(* Logix 5000 project; controller PBS_Perfusion vendor 1 type 14 code 217 rev 32.14; software revision 32.03; part 27 of 27 *)
(* tags used below, declared in another part *)
   AIC703 : P_AInAdv;   // BRX DO PV
   AirManualSP : REAL;
   AirPercentOut : REAL;
   AirProgOper : BOOL;
   AT701 : P_AInAdv;   // DO Transmitter
   AT702 : P_AInAdv;   // pH Transmitter
   BRX_Level_EUMax : REAL;
   BRX_Level_EUmin : REAL;
   BRX_Level_Initialize : BOOL;
   BRX_Level_RawMax : REAL;
   BRX_Level_RawMin : REAL;
   CCAMaxCalc : REAL;
   CO2CVMax : REAL;
   CO2CVMin : REAL;
   CO2EUMax : REAL;
   CO2EUMax_Input : REAL;
   CO2EUMin : REAL;
   CO2EUMin_Input : REAL;
   CO2ManualSP : REAL;
   CO2ManualSP_Input : REAL;
   CO2MaxCalc : REAL;
   CO2PercentOut : REAL;
   CO2ProgOper : BOOL;
   conditionedMedia_auto : BOOL;
   ConditionedMedia_Initialize : BOOL;
   CondMedRawMax : REAL;
   CondMedRawMin : REAL;
   DO_HiDev : REAL;   // hi deviation alarm
   DO_LoDev : REAL;   // low deviation alarm
   DO_ON : BOOL;
   DO_PID_AUTOREQ : BOOL;
   DOPID_INITIALIZE : BOOL;
   EStop : P_DIn;
   FIC110 : P_ValveC;   // PBS CCA
   FIC120 : P_ValveC;   // O2 pbs
   FIC130 : P_ValveC;   // CO2 pbs
   FIC140 : P_ValveC;   // pbs N2 mfc
   GasControl_ON : BOOL;
   GasOffOns : BOOL;
   GasOnOns : BOOL;
   Heater_Output : P_AOut;   // Heating blanket AO
   LIT801 : P_AInAdv;   // Level Value From BRX
   ManualDO_CV : REAL;
   ManualpH_CV : REAL;
   N2CVMax : REAL;
   N2CVMin : REAL;
   N2EUMax : REAL;
   N2EUMax_Input : REAL;
   N2EUMin : REAL;
   N2EUMin_Input : REAL;
   N2ManualSP : REAL;
   N2ManualSP_Input : REAL;
   N2MaxCalc : REAL;
   N2PercentOut : REAL;
   N2ProgOper : BOOL;
   O2CVMax : REAL;
   O2CVMin : REAL;
   O2EUMax : REAL;
   O2EUMax_Input : REAL;
   O2EUMin : REAL;
   O2EUMin_Input : REAL;
   O2ManualSP : REAL;
   O2ManualSP_Input : REAL;
   O2MaxCalc : REAL;
   O2PercentOut : REAL;
   O2ProgOper : BOOL;
   ONS : DINT[3];
   P103 : P_VSD;   // Conditioned Media Addition Pump
   Perfusion_Level_Aggression : REAL;
   pH_HiDev : REAL;   // ph hi deviation
   pH_Initialize : BOOL;
   pH_LoDev : REAL;   // pH Lo deviation alarm
   PH_On : BOOL;
   pH_PID_AUTOREQ : BOOL;
   Temp_Initialize : BOOL;
   TempEUMax : REAL;
   TempEUMin : REAL;
   TempOffOns : BOOL;
   TempOnOns : BOOL;
   TempRawMax : REAL;
   TempRawMin : REAL;
   TotalFlowSP : REAL;
   TT700 : P_AInAdv;   // Temperature Transmitter
   TT700_1Point_Complete : BOOL;
   TT700_1Point_Offset : REAL;
   TT700_2Point_Complete : BOOL;
   TT700_2PointAccept : BOOL;
   TT700_Accept1Point : BOOL;
   TT700_CalClear : BOOL;
   TT700_MaxCfg : REAL;
   TT700_MinCfg : REAL;
   TT700_NewMax : REAL;
   TT700_NewMin : REAL;
   TT700_RawMax : REAL;
   TT700_RawMin : REAL;
   TT700_RawRange : REAL;
   TT700_Ref1Point : REAL;
   TT700_RefMax : REAL;
   TT700_RefMin : REAL;
   TT700_RefRange : REAL;
(* CM_PBS, continued *)

ROUTINE RTD_Calibration   (* ladder *)
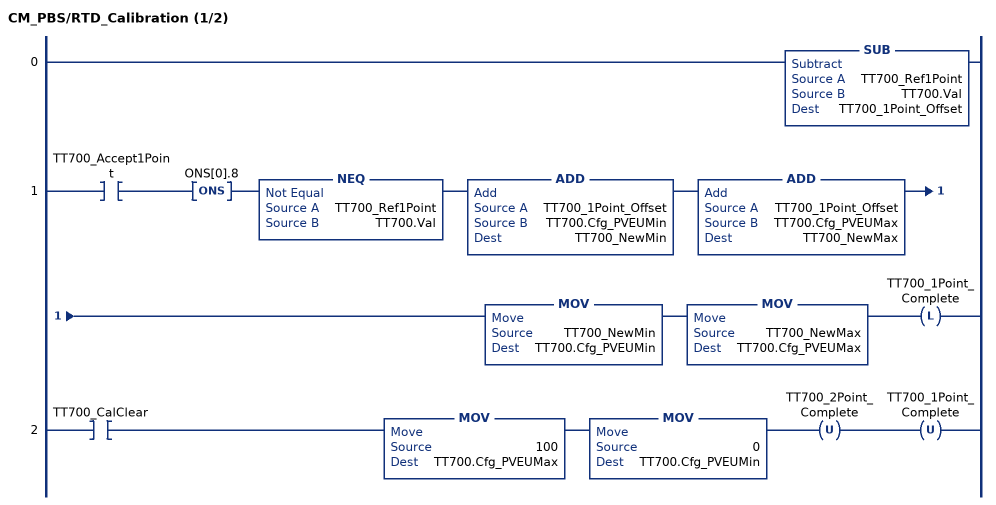
   0: SUB(TT700_Ref1Point,TT700.Val,TT700_1Point_Offset);
   1: XIC(TT700_Accept1Point)ONS(ONS[0].8)NEQ(TT700_Ref1Point,TT700.Val)ADD(TT700_1Point_Offset,TT700.Cfg_PVEUMin,TT700_NewMin)ADD(TT700_1Point_Offset,TT700.Cfg_PVEUMax,TT700_NewMax)MOV(TT700_NewMin,TT700.Cfg_PVEUMin)MOV(TT700_NewMax,TT700.Cfg_PVEUMax)OTL(TT700_1Point_Complete);
   2: XIC(TT700_CalClear)MOV(100,TT700.Cfg_PVEUMax)MOV(0,TT700.Cfg_PVEUMin)OTU(TT700_2Point_Complete)OTU(TT700_1Point_Complete);
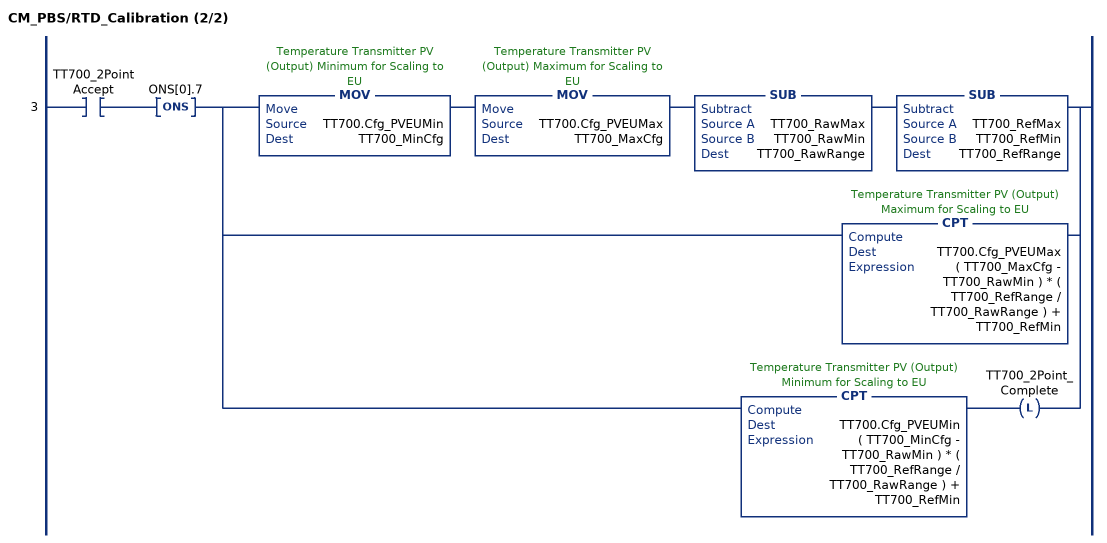
   3: XIC(TT700_2PointAccept)ONS(ONS[0].7)[MOV(TT700.Cfg_PVEUMin,TT700_MinCfg) MOV(TT700.Cfg_PVEUMax,TT700_MaxCfg) SUB(TT700_RawMax,TT700_RawMin,TT700_RawRange) SUB(TT700_RefMax,TT700_RefMin,TT700_RefRange) ,CPT(TT700.Cfg_PVEUMax,( TT700_MaxCfg - TT700_RawMin ) * ( TT700_RefRange / TT700_RawRange ) + TT700_RefMin) ,CPT(TT700.Cfg_PVEUMin,( TT700_MinCfg - TT700_RawMin ) * ( TT700_RefRange / TT700_RawRange ) + TT700_RefMin) OTL(TT700_2Point_Complete) ];
END_ROUTINE
END_PROGRAM

PROGRAM PIDs   (* main routine Main *)
VAR
   ADD_01 : FBD_MATH := (SourceA := 1.0, SourceB := 0.1, Dest := 1.1);
   BOR_01 : FBD_BOOLEAN_OR;
   BOR_02 : FBD_BOOLEAN_OR;
   BOR_03 : FBD_BOOLEAN_OR;
   BOR_04 : FBD_BOOLEAN_OR;
   BOR_05 : FBD_BOOLEAN_OR;
   BOR_06 : FBD_BOOLEAN_OR;
   DIV_01 : FBD_MATH := (SourceA := 10.0, SourceB := 100.0, Dest := 0.1);
   DIV_02 : FBD_MATH := (SourceA := 0.33333334, SourceB := 100.0, Dest := 0.0033333334);
   DIV_03 : FBD_MATH := (SourceB := 100.0);
   DIV_04 : FBD_MATH := (SourceB := 100.0);
   DIV_05 : FBD_MATH := (SourceA := 0.33333334, SourceB := 100.0, Dest := 0.0033333334);
   DIV_06 : FBD_MATH := (SourceA := 0.083333336, SourceB := 100.0, Dest := 0.00083333335);
   DIV_07 : FBD_MATH := (SourceB := 100.0);
   GRT_01 : FBD_COMPARE;
   OSRI_01 : FBD_ONESHOT;
   PIDE_01 : PID_ENHANCED := (PVEUMax := 100.0, SPHLimit := 100.0, RatioProg := 1.0, RatioOper := 1.0, RatioHLimit := 1.0, RatioLLimit := 1.0, CVEUMax := 100.0, CVHLimit := 100.0, PVEDerivative := 1, RTSTime := 1);
   PIDE_02 : PID_ENHANCED := (PVEUMax := 100.0, SPHLimit := 100.0, RatioProg := 1.0, RatioOper := 1.0, RatioHLimit := 1.0, RatioLLimit := 1.0, CVEUMax := 100.0, CVHLimit := 100.0, PVEDerivative := 1, RTSTime := 1);
   PIDE_03 : PID_ENHANCED := (PVEUMax := 100.0, SPHLimit := 100.0, RatioProg := 1.0, RatioOper := 1.0, RatioHLimit := 1.0, RatioLLimit := 1.0, CVEUMax := 100.0, CVHLimit := 100.0, PVEDerivative := 1, RTSTime := 1);
   PIDE_04 : PID_ENHANCED := (PVEUMax := 100.0, SPHLimit := 100.0, RatioProg := 1.0, RatioOper := 1.0, RatioHLimit := 1.0, RatioLLimit := 1.0, CVEUMax := 100.0, CVHLimit := 100.0, PVEDerivative := 1, RTSTime := 1);
   PIDE_05 : PID_ENHANCED := (PVEUMax := 100.0, SPHLimit := 100.0, RatioProg := 1.0, RatioOper := 1.0, RatioHLimit := 1.0, RatioLLimit := 1.0, CVEUMax := 100.0, CVHLimit := 100.0, PVEDerivative := 1, RTSTime := 1);
   SCL_01 : SCALE;
   SUB_01 : FBD_MATH := (SourceA := 1.0, SourceB := 0.1, Dest := 0.9);
END_VAR

ROUTINE GasControl   (* ladder *)
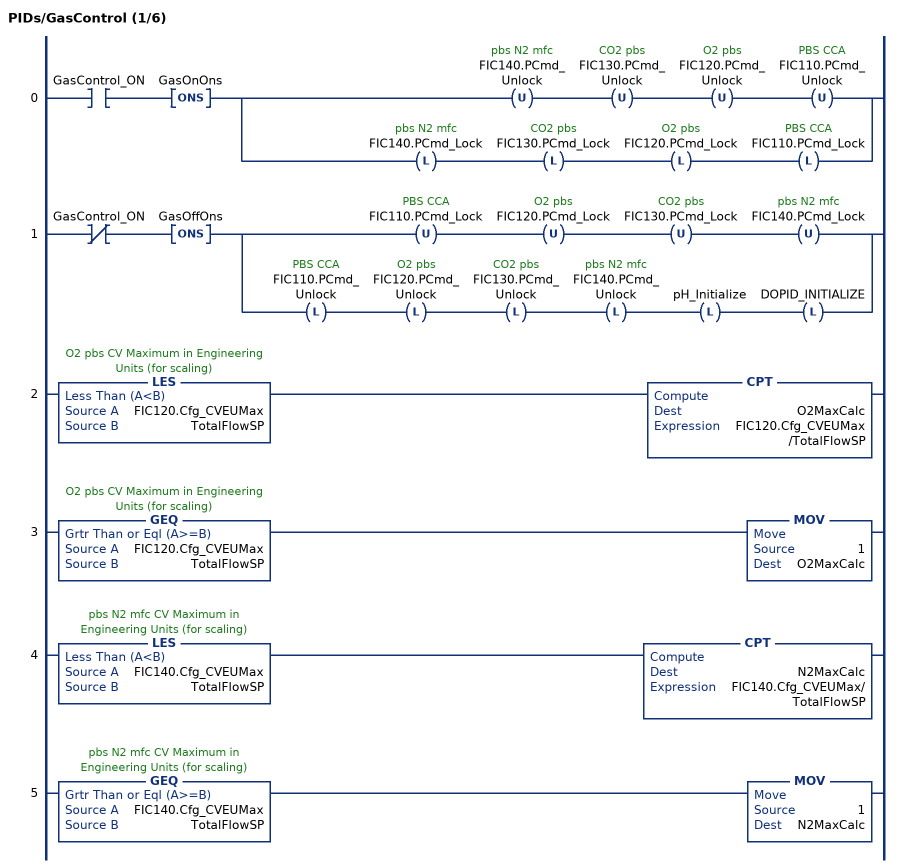
   0: XIC(GasControl_ON)ONS(GasOnOns)[OTU(FIC140.PCmd_Unlock) OTU(FIC130.PCmd_Unlock) OTU(FIC120.PCmd_Unlock) OTU(FIC110.PCmd_Unlock) ,OTL(FIC140.PCmd_Lock) OTL(FIC130.PCmd_Lock) OTL(FIC120.PCmd_Lock) OTL(FIC110.PCmd_Lock) ];
   1: XIO(GasControl_ON)ONS(GasOffOns)[OTU(FIC110.PCmd_Lock) OTU(FIC120.PCmd_Lock) OTU(FIC130.PCmd_Lock) OTU(FIC140.PCmd_Lock) ,OTL(FIC110.PCmd_Unlock) OTL(FIC120.PCmd_Unlock) OTL(FIC130.PCmd_Unlock) OTL(FIC140.PCmd_Unlock) OTL(pH_Initialize) OTL(DOPID_INITIALIZE) ];
   2: LES(FIC120.Cfg_CVEUMax,TotalFlowSP)CPT(O2MaxCalc,FIC120.Cfg_CVEUMax /TotalFlowSP);
   3: GEQ(FIC120.Cfg_CVEUMax,TotalFlowSP)MOV(1,O2MaxCalc);
   4: LES(FIC140.Cfg_CVEUMax,TotalFlowSP)CPT(N2MaxCalc,FIC140.Cfg_CVEUMax/TotalFlowSP);
   5: GEQ(FIC140.Cfg_CVEUMax,TotalFlowSP)MOV(1,N2MaxCalc);
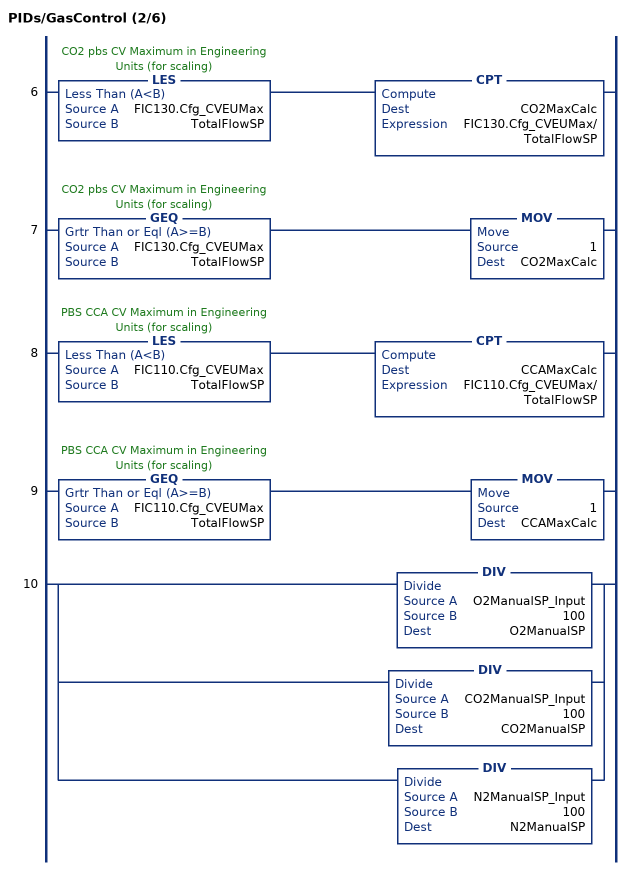
   6: LES(FIC130.Cfg_CVEUMax,TotalFlowSP)CPT(CO2MaxCalc,FIC130.Cfg_CVEUMax/TotalFlowSP);
   7: GEQ(FIC130.Cfg_CVEUMax,TotalFlowSP)MOV(1,CO2MaxCalc);
   8: LES(FIC110.Cfg_CVEUMax,TotalFlowSP)CPT(CCAMaxCalc,FIC110.Cfg_CVEUMax/TotalFlowSP);
   9: GEQ(FIC110.Cfg_CVEUMax,TotalFlowSP)MOV(1,CCAMaxCalc);
   10: [DIV(O2ManualSP_Input,100,O2ManualSP) ,DIV(CO2ManualSP_Input,100,CO2ManualSP) ,DIV(N2ManualSP_Input,100,N2ManualSP) ];
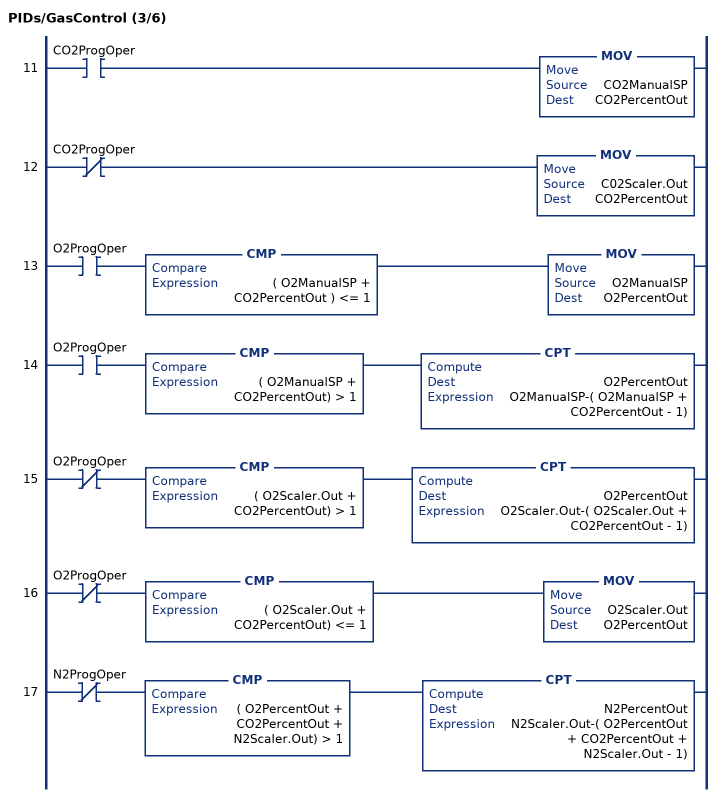
   11: XIC(CO2ProgOper)MOV(CO2ManualSP,CO2PercentOut);
   12: XIO(CO2ProgOper)MOV(C02Scaler.Out,CO2PercentOut);
   13: XIC(O2ProgOper)CMP(( O2ManualSP + CO2PercentOut ) <= 1)MOV(O2ManualSP,O2PercentOut);
   14: XIC(O2ProgOper)CMP(( O2ManualSP + CO2PercentOut) > 1)CPT(O2PercentOut,O2ManualSP-( O2ManualSP + CO2PercentOut - 1));
   15: XIO(O2ProgOper)CMP(( O2Scaler.Out + CO2PercentOut) > 1)CPT(O2PercentOut,O2Scaler.Out-( O2Scaler.Out + CO2PercentOut - 1));
   16: XIO(O2ProgOper)CMP(( O2Scaler.Out + CO2PercentOut) <= 1)MOV(O2Scaler.Out,O2PercentOut);
   17: XIO(N2ProgOper)CMP(( O2PercentOut + CO2PercentOut + N2Scaler.Out) > 1)CPT(N2PercentOut,N2Scaler.Out-( O2PercentOut + CO2PercentOut + N2Scaler.Out - 1));
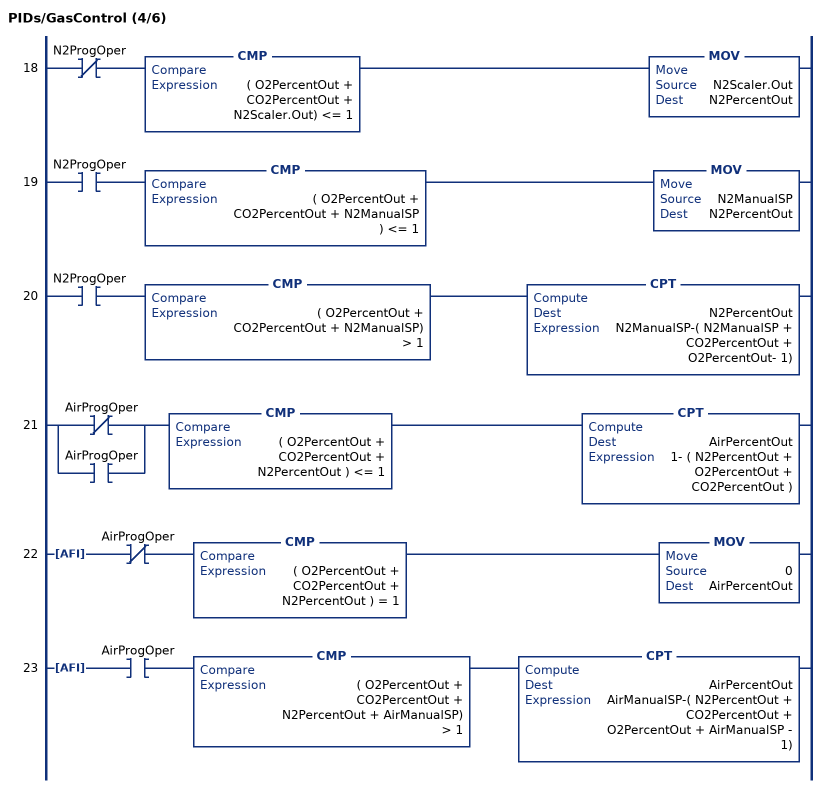
   18: XIO(N2ProgOper)CMP(( O2PercentOut + CO2PercentOut + N2Scaler.Out) <= 1)MOV(N2Scaler.Out,N2PercentOut);
   19: XIC(N2ProgOper)CMP(( O2PercentOut + CO2PercentOut + N2ManualSP ) <= 1)MOV(N2ManualSP,N2PercentOut);
   20: XIC(N2ProgOper)CMP(( O2PercentOut + CO2PercentOut + N2ManualSP) > 1)CPT(N2PercentOut,N2ManualSP-( N2ManualSP + CO2PercentOut + O2PercentOut- 1));
   21: [XIO(AirProgOper) ,XIC(AirProgOper) ]CMP(( O2PercentOut + CO2PercentOut + N2PercentOut ) <= 1)CPT(AirPercentOut,1- ( N2PercentOut + O2PercentOut + CO2PercentOut ));
   22: AFI()XIO(AirProgOper)CMP(( O2PercentOut + CO2PercentOut + N2PercentOut ) = 1)MOV(0,AirPercentOut);
   23: AFI()XIC(AirProgOper)CMP(( O2PercentOut + CO2PercentOut + N2PercentOut + AirManualSP) > 1)CPT(AirPercentOut,AirManualSP-( N2PercentOut + CO2PercentOut + O2PercentOut + AirManualSP - 1));
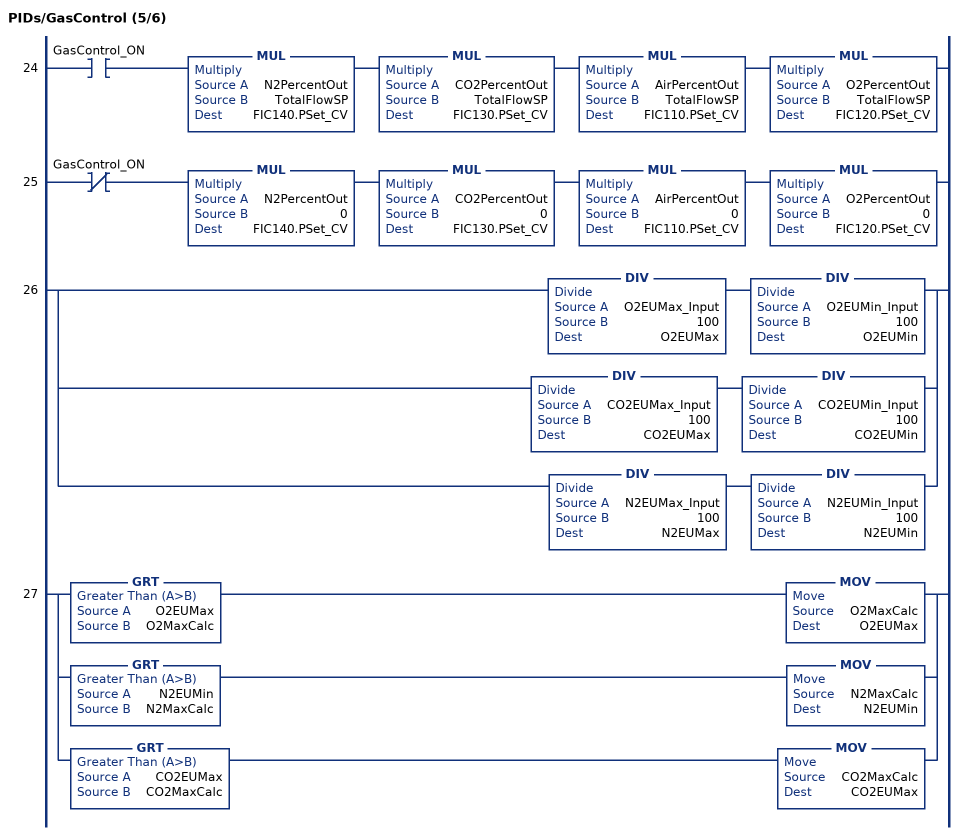
   24: XIC(GasControl_ON)MUL(N2PercentOut,TotalFlowSP,FIC140.PSet_CV)MUL(CO2PercentOut,TotalFlowSP,FIC130.PSet_CV)MUL(AirPercentOut,TotalFlowSP,FIC110.PSet_CV)MUL(O2PercentOut,TotalFlowSP,FIC120.PSet_CV);
   25: XIO(GasControl_ON)MUL(N2PercentOut,0,FIC140.PSet_CV)MUL(CO2PercentOut,0,FIC130.PSet_CV)MUL(AirPercentOut,0,FIC110.PSet_CV)MUL(O2PercentOut,0,FIC120.PSet_CV);
   26: [DIV(O2EUMax_Input,100,O2EUMax) DIV(O2EUMin_Input,100,O2EUMin) ,DIV(CO2EUMax_Input,100,CO2EUMax) DIV(CO2EUMin_Input,100,CO2EUMin) ,DIV(N2EUMax_Input,100,N2EUMax) DIV(N2EUMin_Input,100,N2EUMin) ];
   27: [GRT(O2EUMax,O2MaxCalc) MOV(O2MaxCalc,O2EUMax) ,GRT(N2EUMin,N2MaxCalc) MOV(N2MaxCalc,N2EUMin) ,GRT(CO2EUMax,CO2MaxCalc) MOV(CO2MaxCalc,CO2EUMax) ];
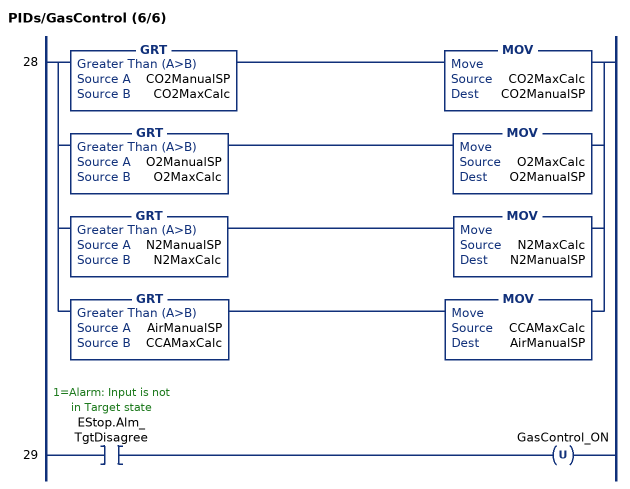
   28: [GRT(CO2ManualSP,CO2MaxCalc) MOV(CO2MaxCalc,CO2ManualSP) ,GRT(O2ManualSP,O2MaxCalc) MOV(O2MaxCalc,O2ManualSP) ,GRT(N2ManualSP,N2MaxCalc) MOV(N2MaxCalc,N2ManualSP) ,GRT(AirManualSP,CCAMaxCalc) MOV(CCAMaxCalc,AirManualSP) ];
   29: XIC(EStop.Alm_TgtDisagree)OTU(GasControl_ON);
END_ROUTINE

ROUTINE Main   (* ladder *)
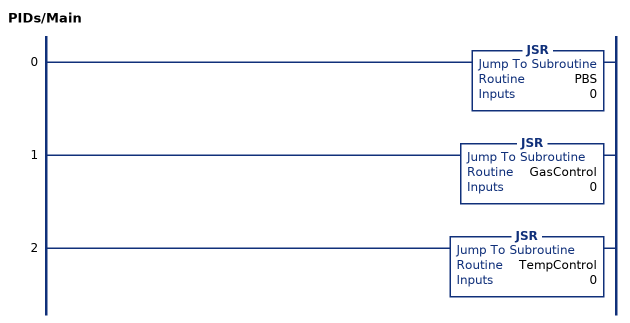
   0: JSR(PBS,0);
   1: JSR(GasControl,0);
   2: JSR(TempControl,0);
END_ROUTINE

ROUTINE PBS   (* function block diagram *)
   SHEET 1
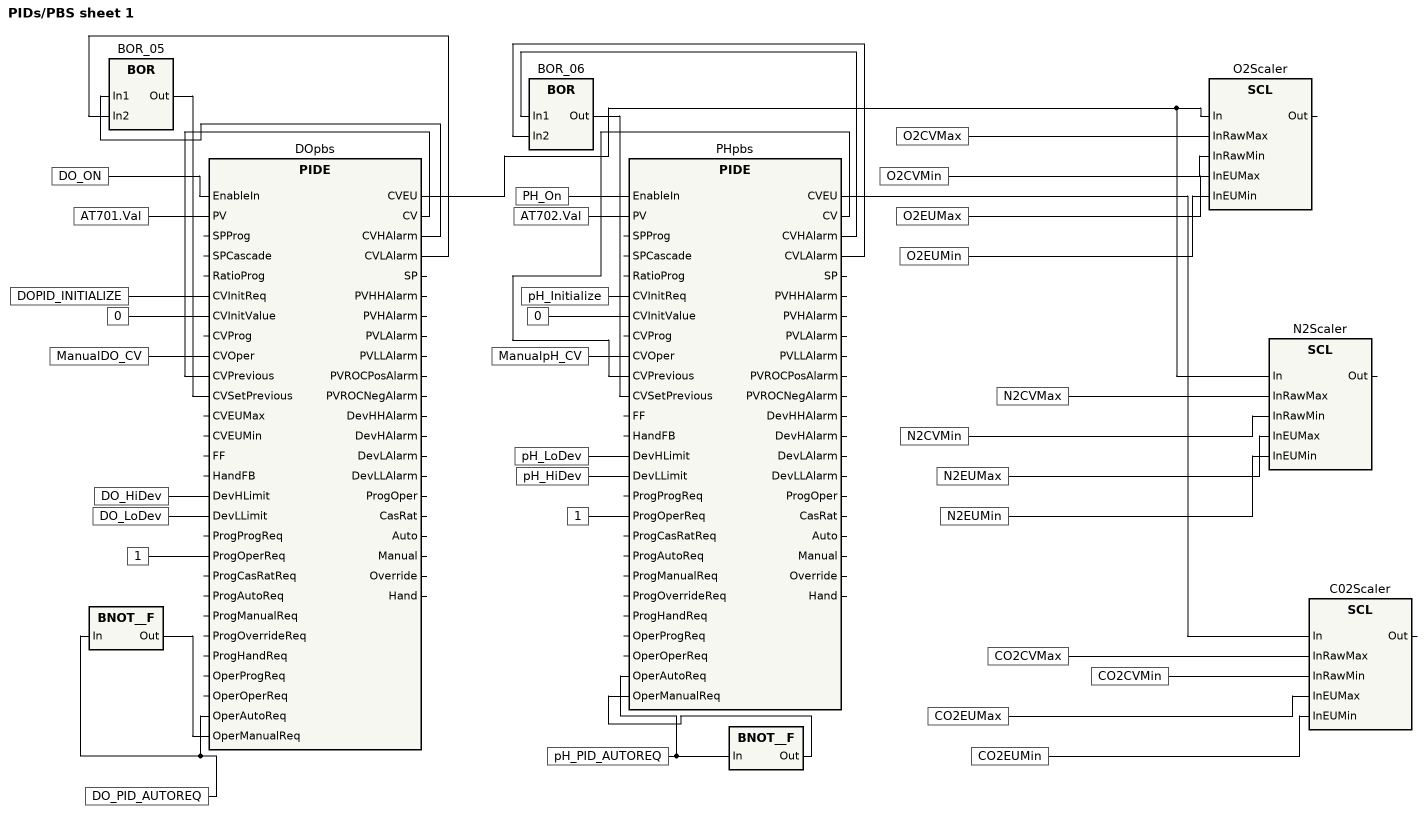
   BOR_05 : BOR(In1 := DOpbs.CVHAlarm {feedback}, In2 := DOpbs.CVLAlarm {feedback});
   BNOT__F_1 : BNOT__F(In := DO_PID_AUTOREQ);
   BOR_06 : BOR(In1 := PHpbs.CVHAlarm {feedback}, In2 := PHpbs.CVLAlarm {feedback});
   BNOT__F_2 : BNOT__F(In := pH_PID_AUTOREQ);
   DOpbs : PIDE(EnableIn := DO_ON, PV := AT701.Val, CVInitReq := DOPID_INITIALIZE, CVInitValue := 0, CVOper := ManualDO_CV, CVPrevious := DOpbs.CV, CVSetPrevious := BOR_05.Out, DevHLimit := DO_HiDev, DevLLimit := DO_LoDev, ProgOperReq := 1, OperAutoReq := DO_PID_AUTOREQ, OperManualReq := BNOT__F_1.Out);   // unwired pins: SPProg SPCascade RatioProg CVProg CVEUMax CVEUMin FF HandFB ProgProgReq ProgCasRatReq ProgAutoReq ProgManualReq ProgOverrideReq ProgHandReq OperProgReq OperOperReq SP PVHHAlarm PVHAlarm PVLAlarm PVLLAlarm PVROCPosAlarm PVROCNegAlarm DevHHAlarm DevHAlarm DevLAlarm DevLLAlarm ProgOper CasRat Auto Manual Override Hand
   O2Scaler : SCL(In := DOpbs.CVEU, InRawMax := O2CVMax, InRawMin := O2CVMin, InEUMax := O2EUMax, InEUMin := O2EUMin);   // unwired pins: Out
   N2Scaler : SCL(In := DOpbs.CVEU, InRawMax := N2CVMax, InRawMin := N2CVMin, InEUMax := N2EUMax, InEUMin := N2EUMin);   // unwired pins: Out
   PHpbs : PIDE(EnableIn := PH_On, PV := AT702.Val, CVInitReq := pH_Initialize, CVInitValue := 0, CVOper := ManualpH_CV, CVPrevious := PHpbs.CV, CVSetPrevious := BOR_06.Out, DevHLimit := pH_LoDev, DevLLimit := pH_HiDev, ProgOperReq := 1, OperAutoReq := pH_PID_AUTOREQ, OperManualReq := BNOT__F_2.Out);   // unwired pins: SPProg SPCascade RatioProg CVProg FF HandFB ProgProgReq ProgCasRatReq ProgAutoReq ProgManualReq ProgOverrideReq ProgHandReq OperProgReq OperOperReq SP PVHHAlarm PVHAlarm PVLAlarm PVLLAlarm PVROCPosAlarm PVROCNegAlarm DevHHAlarm DevHAlarm DevLAlarm DevLLAlarm ProgOper CasRat Auto Manual Override Hand
   C02Scaler : SCL(In := PHpbs.CVEU, InRawMax := CO2CVMax, InRawMin := CO2CVMin, InEUMax := CO2EUMax, InEUMin := CO2EUMin);   // unwired pins: Out
   SHEET 2
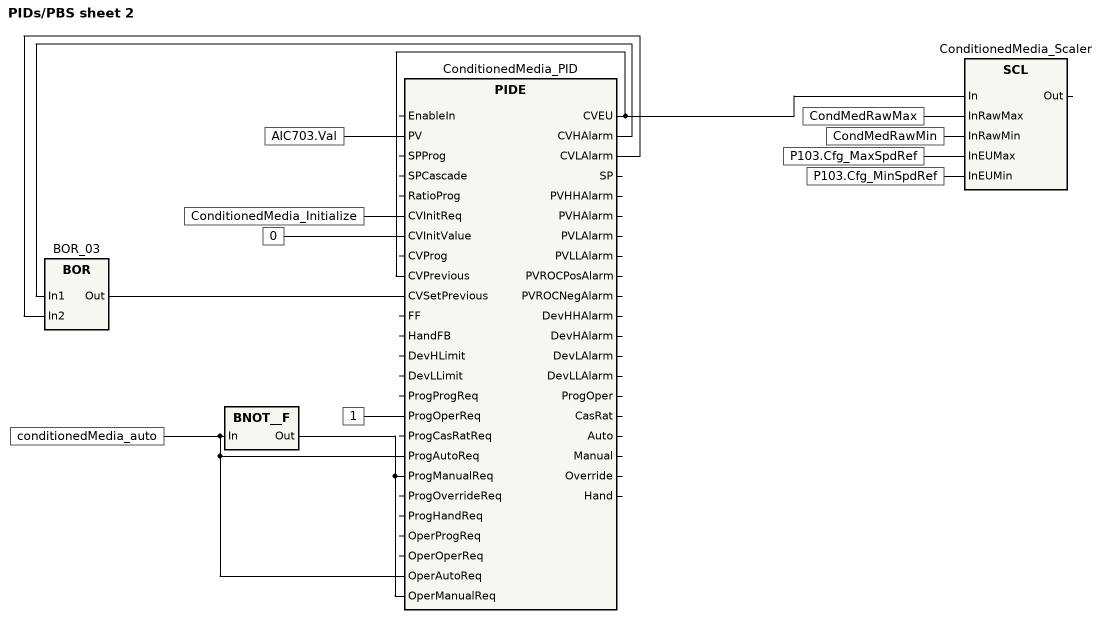
   BOR_03 : BOR(In1 := ConditionedMedia_PID.CVHAlarm {feedback}, In2 := ConditionedMedia_PID.CVLAlarm {feedback});
   BNOT__F_1 : BNOT__F(In := conditionedMedia_auto);
   ConditionedMedia_PID : PIDE(PV := AIC703.Val, CVInitReq := ConditionedMedia_Initialize, CVInitValue := 0, CVPrevious := ConditionedMedia_PID.CVEU, CVSetPrevious := BOR_03.Out, ProgOperReq := 1, ProgAutoReq := conditionedMedia_auto, ProgManualReq := BNOT__F_1.Out, OperAutoReq := conditionedMedia_auto, OperManualReq := BNOT__F_1.Out);   // unwired pins: EnableIn SPProg SPCascade RatioProg CVProg FF HandFB DevHLimit DevLLimit ProgProgReq ProgCasRatReq ProgOverrideReq ProgHandReq OperProgReq OperOperReq SP PVHHAlarm PVHAlarm PVLAlarm PVLLAlarm PVROCPosAlarm PVROCNegAlarm DevHHAlarm DevHAlarm DevLAlarm DevLLAlarm ProgOper CasRat Auto Manual Override Hand
   ConditionedMedia_Scaler : SCL(In := ConditionedMedia_PID.CVEU, InRawMax := CondMedRawMax, InRawMin := CondMedRawMin, InEUMax := P103.Cfg_MaxSpdRef, InEUMin := P103.Cfg_MinSpdRef);   // unwired pins: Out
   SHEET 3
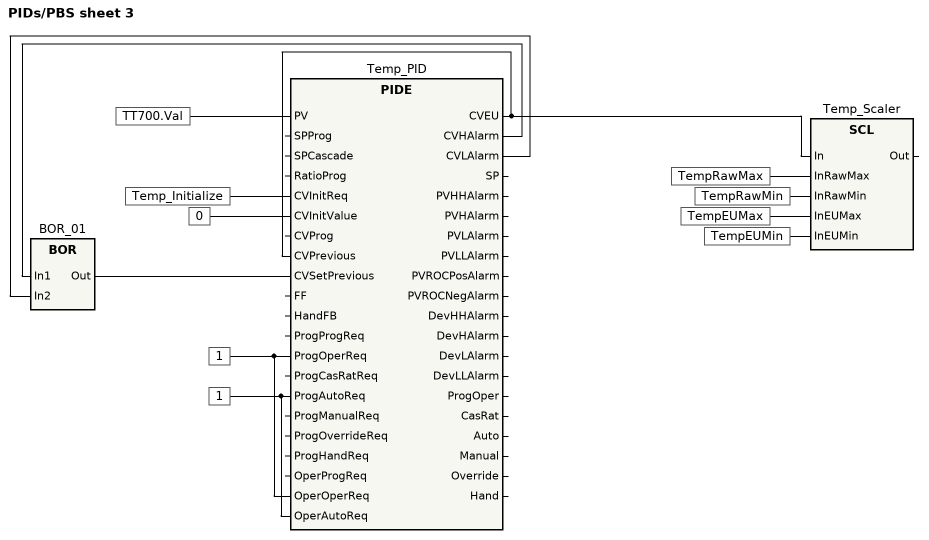
   BOR_01 : BOR(In1 := Temp_PID.CVHAlarm {feedback}, In2 := Temp_PID.CVLAlarm {feedback});
   Temp_PID : PIDE(PV := TT700.Val, CVInitReq := Temp_Initialize, CVInitValue := 0, CVPrevious := Temp_PID.CVEU, CVSetPrevious := BOR_01.Out, ProgOperReq := 1, ProgAutoReq := 1, OperOperReq := 1, OperAutoReq := 1);   // unwired pins: SPProg SPCascade RatioProg CVProg FF HandFB ProgProgReq ProgCasRatReq ProgManualReq ProgOverrideReq ProgHandReq OperProgReq SP PVHHAlarm PVHAlarm PVLAlarm PVLLAlarm PVROCPosAlarm PVROCNegAlarm DevHHAlarm DevHAlarm DevLAlarm DevLLAlarm ProgOper CasRat Auto Manual Override Hand
   Temp_Scaler : SCL(In := Temp_PID.CVEU, InRawMax := TempRawMax, InRawMin := TempRawMin, InEUMax := TempEUMax, InEUMin := TempEUMin);   // unwired pins: Out
   SHEET 4
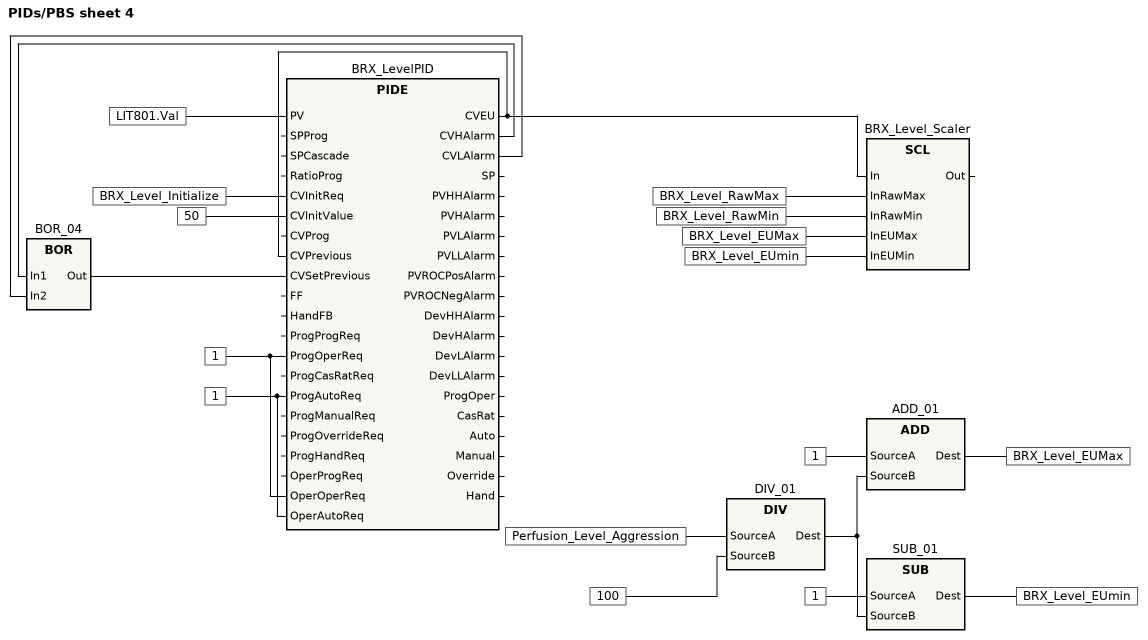
   BOR_04 : BOR(In1 := BRX_LevelPID.CVHAlarm {feedback}, In2 := BRX_LevelPID.CVLAlarm {feedback});
   DIV_01 : DIV(SourceA := Perfusion_Level_Aggression, SourceB := 100);
   ADD_01 : ADD(SourceA := 1, SourceB := DIV_01.Dest);
   SUB_01 : SUB(SourceA := 1, SourceB := DIV_01.Dest);
   BRX_Level_EUMax := ADD_01.Dest;
   BRX_Level_EUmin := SUB_01.Dest;
   BRX_LevelPID : PIDE(PV := LIT801.Val, CVInitReq := BRX_Level_Initialize, CVInitValue := 50, CVPrevious := BRX_LevelPID.CVEU, CVSetPrevious := BOR_04.Out, ProgOperReq := 1, ProgAutoReq := 1, OperOperReq := 1, OperAutoReq := 1);   // unwired pins: SPProg SPCascade RatioProg CVProg FF HandFB ProgProgReq ProgCasRatReq ProgManualReq ProgOverrideReq ProgHandReq OperProgReq SP PVHHAlarm PVHAlarm PVLAlarm PVLLAlarm PVROCPosAlarm PVROCNegAlarm DevHHAlarm DevHAlarm DevLAlarm DevLLAlarm ProgOper CasRat Auto Manual Override Hand
   BRX_Level_Scaler : SCL(In := BRX_LevelPID.CVEU, InRawMax := BRX_Level_RawMax, InRawMin := BRX_Level_RawMin, InEUMax := BRX_Level_EUMax, InEUMin := BRX_Level_EUmin);   // unwired pins: Out
END_ROUTINE

ROUTINE TempControl   (* ladder *)
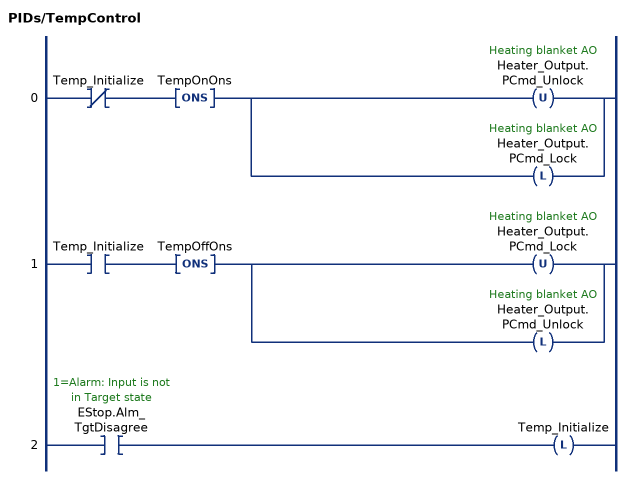
   0: XIO(Temp_Initialize)ONS(TempOnOns)[OTU(Heater_Output.PCmd_Unlock) ,OTL(Heater_Output.PCmd_Lock) ];
   1: XIC(Temp_Initialize)ONS(TempOffOns)[OTU(Heater_Output.PCmd_Lock) ,OTL(Heater_Output.PCmd_Unlock) ];
   2: XIC(EStop.Alm_TgtDisagree)OTL(Temp_Initialize);
END_ROUTINE
END_PROGRAM
